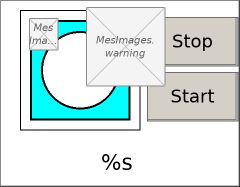
VISUALIZATION VISU_POMPE_CRYO_CTI  // 240x187
VAR_IN_OUT
	m_Input_POMPE:	BLOCK_PCR_CTI_OB;
	m_Input_COM:	BLOCK_RS232_ONBOARD_V4;
	m_Input_Forcage : BOOL;
END_VAR
    Rectangle (0,0 240x187), invisible if: TRUE
    Rectangle (30,20 100x100), colour toggle: m_Input_POMPE.STATE_Ok, invisible if: NOT m_Input_POMPE.State_on
    Rectangle (30,20 100x100), invisible if: NOT m_Input_POMPE.STATE_Ar
    Rectangle (30,20 100x100), invisible if: NOT m_Input_POMPE.STATE_Regen
    Group (41,31 78x78)
        Ellipse (0,0 78x78)
        Polyline (25,37)
        Polyline (10,4)
        Polyline (18,14)
        Polyline (26,37)
        Polyline (25,38)
    Rectangle (20,10 120x120), invisible if: NOT (m_Input_POMPE.AUTOR_On_IHM OR m_Input_POMPE.AUTOR_Off_IHM) OR NOT PRG_User.ACTU_USER.MAINTENANCE
        tap m_Input_POMPE.M_ON
    Rectangle (98,140 140x45), "%s", text variable: m_Input_POMPE.MNEMO
    Button (147,17 91x49), "Regen", invisible if: NOT m_Input_POMPE.AUTOR_Regen_IHM OR NOT PRG_User.ACTU_USER.MAINTENANCE OR m_Input_POMPE.STATE_Regen
        toggle m_Input_POMPE.M_Regen
    Button (147,17 91x49), "Stop", invisible if: NOT PRG_User.ACTU_USER.MAINTENANCE OR NOT m_Input_POMPE.STATE_Regen
        OnMouseDown: execute { m_Input_COM.CO_StopRegen:=TRUE; }
        OnMouseUp: execute { m_Input_COM.CO_StopRegen:=FALSE; }
    Button (147,72 91x49), "Start", invisible if: NOT PRG_User.ACTU_USER.MAINTENANCE OR NOT m_Input_POMPE.OUT_On OR ( NOT m_Input_COM.STATE_Pompe = 0) OR m_Input_POMPE.STATE_Regen
        OnMouseDown: execute { m_Input_Forcage:=TRUE; }
        OnMouseUp: execute { m_Input_Forcage:=FALSE; }
    Image (86,7 79x79), invisible if: NOT m_Input_POMPE.STATE_NOK, image: MesImages.warning
    Image (29,18 29x32), invisible if: NOT m_Input_COM.STATE_Pompe, image: MesImages.Flocon
END_VISUALIZATION

(* stored: Version 1.1.0.1, ProductVersion 3.1.4026.18
   Visu VISU_POMPE_CRYO_CTI: Id {3f2da4dc-e1aa-4927-a393-2df99b64fec4} *)
